FUNCTION_BLOCK LinearContinuousDrive_3Sensor EXTENDS FBA_LinearDrive IMPLEMENTS I_LinearContinuousDrive
VAR_INPUT
	drive : I_ContinuousDrive;
	allowDualSideTraverse : BOOL; //allows motion between home to retractLimit
END_VAR
VAR
	extendLimit AT %I* : BOOL;
	retractLimit AT %I* : BOOL;
END_VAR

override();

ready := bEnable AND NOT Active AND HomeSet;

PROPERTY Active : BOOL
GET
Active := drive.Active;
END_GET
END_PROPERTY

PROPERTY AtExtendLimit : BOOL
GET
AtExtendLimit := extendLimit <> sensorDefaultState;
END_GET
END_PROPERTY

PROPERTY AtRetractLimit : BOOL
GET
AtRetractLimit := retractLimit <> sensorDefaultState;
END_GET
END_PROPERTY

PROPERTY Error : BOOL
GET
error := drive.Error;
END_GET
END_PROPERTY

METHOD homingSequence : BOOL
(*
homing sequence is different for linear motion devices with limit sensors
*)
CASE step OF
	Homing.IDLE:
		reset();
		IF bEnable THEN
			step := Homing.RETRY;
		END_IF
		
	Homing.START:
		IF AtHome THEN
			step := Homing.STOP;
			
		ELSIF AtRetractLimit THEN
			step := Homing.RETRY;
			
		ELSE
			moveContinuous(newDirection:= MC_Positive_Direction);
		END_IF
		
	Homing.RETRY:
		IF AtExtendLimit THEN
			step := Homing.START;
		ELSE
			moveContinuous(newDirection:= MC_Positive_Direction);
		END_IF
		
	Homing.STOP:
		IF stop() THEN
			step := Homing.DONE;
		END_IF
		
	Homing.DONE:
		homingComplete := TRUE;
		step := Homing.IDLE;
		
END_CASE
END_METHOD

METHOD moveContinuous : BOOL
VAR_INPUT
	newDirection : MC_Direction;
END_VAR
drive.moveContinuous(newDirection:= newDirection);

direction := newDirection;
END_METHOD

METHOD PRIVATE override : BOOL
VAR_INPUT
END_VAR
(*
-at home and attempting to traverse outward
-at outer limit and attempting to traverse outward
-at inner limit and attempting to traverse inwards
*)
(*
inward = negative direction, negative velocity
outward = positive direction, positive velocity
*)

IF error THEN
	stop();
	reset();
	
ELSIF
	(NOT allowDualSideTraverse AND AtHome AND direction = MC_Positive_Direction) OR
	(AtExtendLimit AND direction = MC_Negative_Direction) OR
	(AtRetractLimit AND direction = MC_Positive_Direction)
THEN
	stop();
END_IF
END_METHOD

METHOD reset : BOOL
VAR_INPUT
END_VAR
reset := drive.reset();
END_METHOD

METHOD stop : BOOL
VAR_INPUT
END_VAR
stop := drive.stop();
END_METHOD

METHOD toHome : BOOL
VAR_INPUT
END_VAR
IF AtHome THEN
	toHome := TRUE;
ELSE
	moveContinuous(newDirection := MC_Negative_Direction);
END_IF
END_METHOD

END_FUNCTION_BLOCK

(* stored: Version 1.1.0.1, ProductVersion 3.1.4024.11
   POU LinearContinuousDrive_3Sensor: Id {c13fdb69-1504-4b8b-bb33-c0c733ab430a}, SpecialFunc None
   Folder Private: Id {6de7fe8d-38f4-4558-877b-899f1f6f8f4d}
   Folder Properties: Id {2d4d85ee-a6c1-4363-9b96-3ff8256abc4a}
   Property Active: Id {999cdb38-6a9a-40bf-ab33-71e84dcc1fd0}
   Get Get: Id {a2c211dd-f7b4-44b4-b2f6-0020a2a0a655}
   Property AtExtendLimit: Id {bd0dba66-91bc-4de0-9418-fa30f53e8e25}
   Get Get: Id {23cdf262-7aec-4560-870e-b643bf7ac6be}
   Property AtRetractLimit: Id {f16bd607-997c-484e-afe3-fd8fc3eeeb9f}
   Get Get: Id {cb98346f-33c4-4e80-9193-80e8da7ebe88}
   Property Error: Id {51c01f70-9a54-4c17-bf32-d68c79a458cf}
   Get Get: Id {230db7a3-5116-487c-97f1-758523510e7c}
   Method homingSequence: Id {8cd879a5-4ac9-444d-a242-18853a4ba174}
   Method moveContinuous: Id {ff282c40-4c0a-4ab0-97ff-6384ddf92b60}
   Method override: Id {5d022c1d-b087-4cc8-b413-18ebc5f9d5e3}
   Method reset: Id {6ba26e74-3166-430f-b9c6-7c13714be874}
   Method stop: Id {ff999892-3f4d-48a2-bfab-964ee6079f09}
   Method toHome: Id {9f64872e-7516-4c4e-acd0-088f56e0cad1} *)
